FUNCTION_BLOCK Z_TEMPERATURE (* Basic FB with empty ECC *)
  (* Standard: 61499-2 *)
  (* Version 1.0, 2020-10-20, chong *)
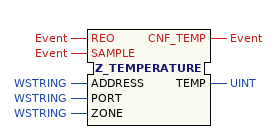
  EVENT_INPUT
    REO;
    SAMPLE;
  END_EVENT
  EVENT_OUTPUT
    CNF_TEMP;
  END_EVENT
  VAR_INPUT
    ADDRESS : WSTRING;
    PORT : WSTRING;
    ZONE : WSTRING;
  END_VAR
  VAR_OUTPUT
    TEMP : UINT;
  END_VAR
  VAR
    INTERNALVAR1 : BOOL; (* Internal Variable *)
    INTERNALVAR2 : BOOL; (* Internal Variable *)
  END_VAR
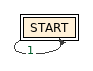
  EC_STATES
    START; (* Initial State *)
  END_STATES
  EC_TRANSITIONS
    START TO START := 1;
  END_TRANSITIONS
  ALGORITHM ALG1 IN ST: (* New Algorithm *)

  END_ALGORITHM
  ALGORITHM ALG2 IN ST: (* New Algorithm *)

  END_ALGORITHM
  ALGORITHM ALG3 IN ST: (* New Algorithm *)

  END_ALGORITHM
  SERVICE left interface/right interface (* Basic FB with empty ECC *)
    SEQUENCE Service Sequence
      left interface.INIT();
      -> left interface.INITO() -> right interface.INITO();
    END_SEQUENCE
  END_SERVICE
END_FUNCTION_BLOCK
